(* IEC 61131-3 sources: inproshop/test13_exported/1.Function/FB/ElectricScrewdriver(电批), 6 files *)

(* ---- Str_ESD.st ---- *)
TYPE Str_ESD :
STRUCT
	Cmd:Str_ESDCmd;//控制
	Parm:Str_ESDParm;//参数
	Status:Str_ESDStatus;//状态
	DevStatus:Str_ESDDevStatus;//硬件IO映射
END_STRUCT
END_TYPE

(* ---- Str_ESDCmd.st ---- *)
TYPE Str_ESDCmd :
STRUCT
	Power	:BOOL;//使能
	Stop	:BOOL;//停止
	AutoStart:BOOL;//自动启动
	ManuStart:BOOL;//手动启动
	AutoFoward	:BOOL;//自动正转
	AutoBackward	:BOOL;//自动反转
	ManuFoward	:BOOL;//手动正转
	ManuBackward	:BOOL;//手动反转

END_STRUCT
END_TYPE

(* ---- Str_ESDDevStatus.st ---- *)
TYPE Str_ESDDevStatus :
STRUCT
	iNG:BOOL;//锁附NG
	iOK:BOOL;//锁附OK
	iERROR:BOOL;//电批报警
	oPowerOn:BOOL;//电批使能
	oStart:BOOL;//电批启动
	oReset:BOOL;//报警复位
END_STRUCT
END_TYPE

(* ---- Str_ESDParm.st ---- *)
TYPE Str_ESDParm :
STRUCT
	Velocity	:INT;//控制速度
	Torque	:INT;//控制扭矩
	GoalNum:INT := 1;//锁螺丝目标数量
    Velocity1	:INT;//控制速度1
	Torque1	:INT;//控制扭矩1
	Velocity2	:INT;//控制速度2
	Torque2	:INT;//控制扭矩2
END_STRUCT
END_TYPE

(* ---- Str_ESDStatus.st ---- *)
TYPE Str_ESDStatus :
STRUCT
	PowerON	:BOOL;//电批已使能
	Busy	:BOOL;//锁附中
	PosOK	:BOOL;//锁附完成
	OK	:BOOL;//锁附OK
	NG	:BOOL;//锁附NG
	VolNum:INT;//锁螺丝当前数量
	Error	:BOOL;//错误
	ErrorID	:WORD;//错误代码
	SpTime		:UINT;//锁附时间
	State		:INT;//电批状态=1锁附中,=2锁附OK,=3锁附NG
END_STRUCT
END_TYPE

(* ---- FB_ElectricScrewdriver_V1_1_0.st ---- *)
FUNCTION_BLOCK FB_ElectricScrewdriver_V1_1_0
VAR_IN_OUT
	ioESDCtrl:Str_ESD;
END_VAR

VAR_INPUT
	iName:WSTRING(40);//轴名称
	iEstop:BOOL;//急停
	iSafeDoor:BOOL;//安全门信号
	iLightCurtain:BOOL;//光栅信号
	iMode:Str_Mode;//设备模式
	iNG:BOOL;//锁附NG
	iOK:BOOL;//锁附OK
	iERROR:BOOL;//电批报警
END_VAR
VAR_OUTPUT
	oPowerOn:BOOL;//电批使能
	oStart:BOOL;//电批启动
	oReset:BOOL;//报警复位
END_VAR
VAR
	i:INT;//循环数据用
	En_Control:BOOL;//轴控制条件
	StartDelay:TON;//启动计时
END_VAR
VAR RETAIN PERSISTENT
	// 启动计时
	Velocity: INT;
	Torque:INT;
END_VAR

(*版本V1:
	功能块建立
*)

IF CPU_Clock.FirstRun THEN
	ioESDCtrl.Parm.Velocity:=Velocity;
	ioESDCtrl.Parm.Torque:=Torque;
ELSE
	Velocity:=ioESDCtrl.Parm.Velocity;
	Torque:=ioESDCtrl.Parm.Torque;
END_IF

//初始值赋值
//速度
IF ioESDCtrl.Parm.Velocity<=0 THEN
	ioESDCtrl.Parm.Velocity:=100;
END_IF
//扭矩
IF ioESDCtrl.Parm.Torque<=0 THEN
	ioESDCtrl.Parm.Torque:=100;
END_IF

//自动模式下自动使能
IF iMode.Status.AutoMode THEN
	ioESDCtrl.Cmd.Power:=TRUE;
END_IF

//使能
oPowerOn:= iEstop AND iSafeDoor AND iLightCurtain AND ioESDCtrl.Cmd.Power;

//控制
IF iMode.Status.AutoMode THEN
	oStart:=ioESDCtrl.Cmd.AutoStart;
ELSIF iMode.Status.ManualMode THEN
	oStart:=ioESDCtrl.Cmd.ManuStart;
END_IF

//信号转换
IF oStart THEN
	IF iOK THEN
		ioESDCtrl.Status.OK:=TRUE;
	ELSIF iNG OR StartDelay.Q THEN
		ioESDCtrl.Status.NG:=TRUE;
	END_IF
ELSE
	ioESDCtrl.Status.OK:=FALSE;
	ioESDCtrl.Status.NG:=FALSE;
END_IF

//急停
IF NOT iEstop THEN
	oStart:=FALSE;
END_IF

StartDelay(IN:= oStart, PT:= T#30S, Q=> , ET=> );

//切换模式手动清除信号
IF iMode.Status.AutoMode THEN
	ioESDCtrl.Cmd.ManuBackward:=FALSE;
	ioESDCtrl.Cmd.ManuFoward:=FALSE;
	ioESDCtrl.Cmd.ManuStart:=FALSE;
END_IF
//自复位自动控制信号
ioESDCtrl.Cmd.AutoBackward:=FALSE;
ioESDCtrl.Cmd.AutoFoward:=FALSE;
ioESDCtrl.Cmd.AutoStart:=FALSE;
